// TIA Portal project "queue_of_items_counter_plc" (V19)
// Vorlageprojekt für das Buch mit Zielsystem S7-1200

(* hardware
DEVICE "S7-1200-Station_1"  S7-1200 Station
   slot 0: "Baugruppenträger_0"  Rack  V1.0
   slot 1: "PLC_1"  CPU 1211C DC/DC/DC  6ES7 211-1AE40-0XB0  V4.1
*)

// ===== PLC "PLC_1"  CPU 1211C DC/DC/DC =====

VAR_GLOBAL   // PLC tag table "Standard-Variablentabelle"
   "buffer_conveyor" AT %Q0.1 : Bool;
   "start" AT %E0.0 : Bool;
   "ready_sensor" AT %E0.1 : Bool;
   "entry_sensor" AT %I0.2 : Bool;
   "exit_sensor" AT %I0.3 : Bool;
   "entry_conveyor" AT %Q0.0 : Bool;
   "entry_conveyor_flag" AT %M0.0 : Bool;
   "buffer_conveyor_flag" AT %M0.1 : Bool;
   "exit_sensor_off_detect" AT %M0.4 : Bool;
   "ready_sensor_off_detect" AT %M0.2 : Bool;
   "entry_sensor_off_detect" AT %M0.3 : Bool;
   "reset" AT %I0.4 : Bool;
   "start_detect" AT %M0.5 : Bool;
   "reset_detect" AT %M0.6 : Bool;
END_VAR

// folder: System blocks/Program resources

DATA_BLOCK "entry_counter"   // DB2
{ S7_Optimized_Access := 'TRUE' }
AUTHOR : Simatic
FAMILY : IEC
NAME : CNTR
VERSION : 1.0
// stored: InstanceOfName IEC_COUNTER
"IEC_COUNTER"
BEGIN
END_DATA_BLOCK

DATA_BLOCK "ready_counter"   // DB3
{ S7_Optimized_Access := 'TRUE' }
AUTHOR : Simatic
FAMILY : IEC
NAME : CNTR
VERSION : 1.0
// stored: InstanceOfName IEC_COUNTER
"IEC_COUNTER"
BEGIN
END_DATA_BLOCK

DATA_BLOCK "exit_counter"   // DB5
{ S7_Optimized_Access := 'TRUE' }
AUTHOR : Simatic
FAMILY : IEC
NAME : CNTR
VERSION : 1.0
// stored: InstanceOfName IEC_COUNTER
"IEC_COUNTER"
BEGIN
END_DATA_BLOCK

// folder: (top level)

FUNCTION "MHJ-PLC-Lab-Function-S71200" : Void   // FC9000, SCL
{ S7_Optimized_Access := 'TRUE' }
VERSION : 0.1
   VAR_TEMP
      rdTimeReturn : Int;
      outputTime : DTL;
      SyncVal : Byte;
      forVal : Int;
      forVal_2 : Int;
      Value : Byte;
   END_VAR
   VAR CONSTANT
      CompVal : Byte := 16#34;
      Value_01 : Byte := 16#11;
      Value_01_DW : DWord := 16#A165_D992;
      Value_02_DW : DWord := 16#58BE_4401;
   END_VAR
BEGIN

   #Value:=PEEK(area := 16#82,
        dbNumber := 0,
        byteOffset := 511);
   #Value := #Value + 1;

   POKE(area := 16#82,
        dbNumber := 0,
        byteOffset := 511,
        value := #Value);

   POKE(area:=16#81,
        dbNumber:=0,
        byteOffset:=1016,
        value:=#Value_01_DW);
   POKE(area := 16#81,
        dbNumber := 0,
        byteOffset := 1020,
        value := #Value_02_DW);

   POKE(area := 16#81,
        dbNumber := 0,
        byteOffset := 511,
        value := B#16#00);

   FOR #forVal := 0 TO 120 DO
       FOR #forVal_2:=0 TO 10 DO
           #rdTimeReturn:=RD_SYS_T(#outputTime);
           #rdTimeReturn := WR_SYS_T(#outputTime);
           #rdTimeReturn := RD_SYS_T(#outputTime);
           #rdTimeReturn := WR_SYS_T(#outputTime);
       END_FOR;
       #SyncVal:= PEEK(area := 16#81,
                      dbNumber := 0,
                      byteOffset := 511);
       IF #SyncVal = #CompVal THEN
          GOTO M_1;
       END_IF;
   END_FOR;
   RETURN;

   M_1:
   POKE(area := 16#81,
        dbNumber := 0,
        byteOffset := 511,
        value := B#16#0);
END_FUNCTION

ORGANIZATION_BLOCK "Main"   // OB1, FBD, ProgramCycle
TITLE = "Main Program Sweep (Cycle)"
{ S7_Optimized_Access := 'TRUE' }
VERSION : 0.1
   VAR_INPUT
      Initial_Call : Bool;   // Initial call of this OB
      Remanence : Bool;   // =True, if remanent data are available
   END_VAR
BEGIN

REGION Network 1: Konnektierungsbaustein für PLC-Lab
   // Im Netzwerk 1 wird der Konnektierungsbaustein für PLC-Lab aufgerufen.
   // Dieser Aufruf darf nicht entfernt werden!
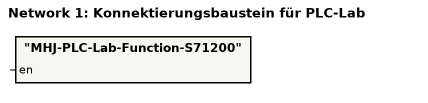
   "MHJ-PLC-Lab-Function-S71200"();
END_REGION

REGION Network 2: Ihr Programm
   // Schreiben Sie ab Netzwerk 2 Ihr Programm
END_REGION
END_ORGANIZATION_BLOCK

ORGANIZATION_BLOCK "Main_1"   // OB123, LAD, ProgramCycle
TITLE = "Main Program Sweep (Cycle)"
{ S7_Optimized_Access := 'TRUE' }
VERSION : 0.1
   VAR_INPUT
      Initial_Call : Bool;   // Initial call of this OB
      Remanence : Bool;   // =True, if remanent data are available
   END_VAR
   VAR_TEMP   // added for the SCL form of the ladder/FBD networks
      _w1 : Bool;
   END_VAR
BEGIN

REGION Network 1
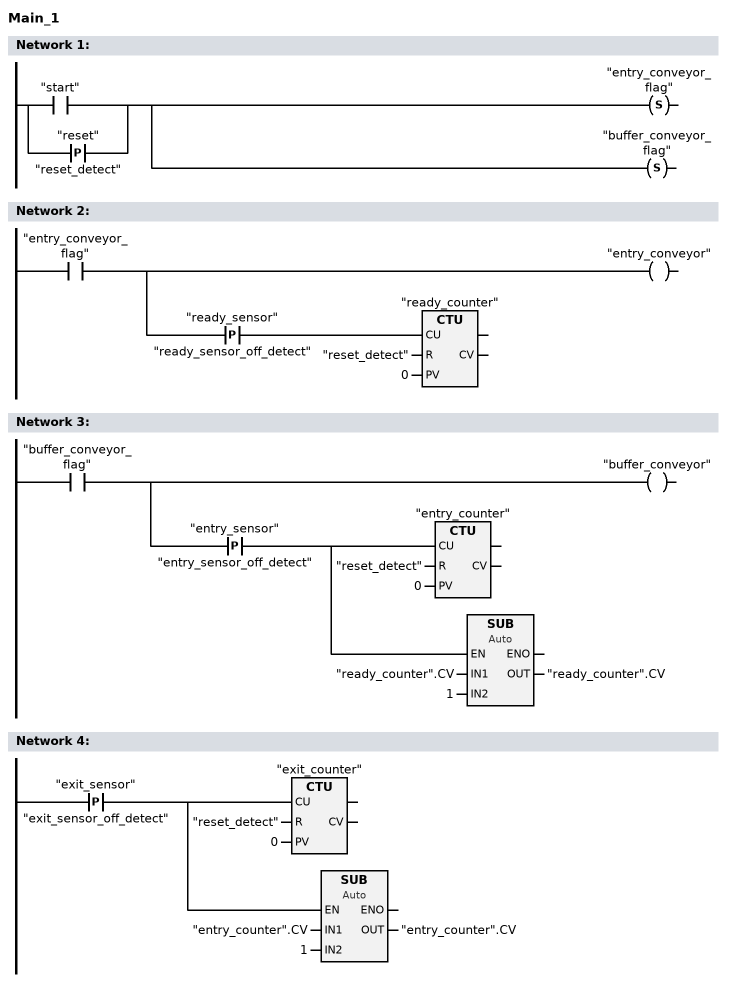
   RUNG wire#powerrail
      Contact( "start" )
      wire#w1
      S_Coil( "entry_conveyor_flag" )
   END_RUNG
   RUNG wire#powerrail
      P_Contact(operand := "reset", bit := "reset_detect")
   END_RUNG wire#w1
   RUNG wire#w1
      S_Coil( "buffer_conveyor_flag" )
   END_RUNG
   // the same network as SCL:
   #_w1 := "reset" AND NOT "reset_detect";   // rising edge of "reset"
   "reset_detect" := "reset";
   IF "start" OR #_w1 THEN
       "entry_conveyor_flag" := TRUE;
       "buffer_conveyor_flag" := TRUE;
   END_IF;
END_REGION

REGION Network 2
   "entry_conveyor" := "entry_conveyor_flag";
   #_w1 := "entry_conveyor_flag" AND "ready_sensor" AND NOT "ready_sensor_off_detect";   // rising edge of "ready_sensor"
   "ready_sensor_off_detect" := "ready_sensor";
   "ready_counter".CTU(CU := #_w1, R := "reset_detect", PV := 0);
END_REGION

REGION Network 3
   "buffer_conveyor" := "buffer_conveyor_flag";
   #_w1 := "buffer_conveyor_flag" AND "entry_sensor" AND NOT "entry_sensor_off_detect";   // rising edge of "entry_sensor"
   "entry_sensor_off_detect" := "entry_sensor";
   "entry_counter".CTU(CU := #_w1, R := "reset_detect", PV := 0);
   IF #_w1 THEN "ready_counter".CV := "ready_counter".CV - 1; END_IF;
END_REGION

REGION Network 4
   #_w1 := "exit_sensor" AND NOT "exit_sensor_off_detect";   // rising edge of "exit_sensor"
   "exit_sensor_off_detect" := "exit_sensor";
   "exit_counter".CTU(CU := #_w1, R := "reset_detect", PV := 0);
   IF #_w1 THEN "entry_counter".CV := "entry_counter".CV - 1; END_IF;
END_REGION
END_ORGANIZATION_BLOCK